PROGRAM Z_CIRC

(*-------------------------------------------------------------------------------------------------------*)

(*v042 Ev. Intercepta Salida Bomba*)

MC._08_CIRC.v042_OutPump.xOpen:= F_VACIADO.z_CloseCuttingV;

(*v044 Ev. Spray*)
MC._08_CIRC.v044_Spray.xOpen:= F_DUCHAS.Z_Spray;

END_PROGRAM

(* stored: Version 1.1.0.1, ProductVersion 3.1.4024.10
   POU Z_CIRC: Id {3ae77c83-523f-48c1-a6aa-a4978d7e8d00}, SpecialFunc None *)
